Staubli VAL3: production.dtx

num nEvent
num nKey = 255
num nMax
num nMin
public num nPage
num nPoint
num nRefresh
num nTime = 5
public num nToSuperV
num nValue
num nIndex
num nSelect
num nView
num nClockScroll
num nFile
string sEvent
public string sItems
string sMenu[4]
  [0] = "HOME"
  [1] = "Emap"
  [2] = "Pallet"
  [3] = "Process"
string sMenu8[8]
string sMessage
string sLogAction
bool bButton[8]
  [0] = true
  [1] = true
  [2] = true
  [3] = true
  [6] = true
bool bLarge
bool bPage
bool bRefreshPoint = true
bool bRefreshProg
bool bShowMessage
bool bTrajLoad
bool bShowInit
bool bUseAutoScroll
num nPointLine[200]
string sProgName
string sTrajName
bool bTraj
